KUKA KRL program: G1_Prog.src, G1_Prog.dat

--- G1_Prog.src ---
&ACCESS RVP
DEF  G1_Prog ( )

   GLOBAL INTERRUPT DECL 3 WHEN $STOPMESS==TRUE DO IR_STOPM ( )
   INTERRUPT ON 3
   BAS (#INITMOV,0 )
   BAS (#TOOL, XTOOL)
   BAS (#BASE, XTOOLBASE)

 ;Mover PARA HOME
   SPTP XHOME
   LOOP
      PLC_GET_Pos()
      Gridplace()
      SPTP XHOME
   ENDLOOP

END

DEF PLC_GET_Pos()
   WAIT FOR $IN[19]
   WAIT FOR NOT $IN[19]
   NextPos = 0

   IF $IN[19]THEN
      NextPos=NextPos+1
   ENDIF
   IF $IN[20]THEN
      NextPos=NextPos+2
   ENDIF
   IF $IN[21]THEN
      NextPos=NextPos+4
   ENDIF
   IF $IN[22]THEN
      NextPos=NextPos+8
   ENDIF
END

DEF Gridplace()
   SWITCH NextPos
      CASE 0
         ;insert your code here
         MoveTo(Matrix_Pos1)
      CASE 1
         ;insert your code here
         MoveTo(Matrix_Pos2)
      CASE 2
         ;insert your code here
         MoveTo(Matrix_Pos3)
      CASE 3
         ;insert your code here
         MoveTo(Matrix_Pos4)
      CASE 4
         ;insert your code here
         MoveTo(Matrix_Pos5)
      CASE 5
         ;insert your code here
         MoveTo(Matrix_Pos6)
      CASE 6
         ;insert your code here
         MoveTo(Matrix_Pos7)
      CASE 7
         ;insert your code here
         MoveTo(Matrix_Pos8)
      CASE 8
         ;insert your code here
         MoveTo(Matrix_Pos9)
      DEFAULT
         ;insert your code here
   ENDSWITCH
END

DEF MoveTo(Position:IN)
 POS Position
 RECOLHA.C = 0
 Position.C = 0

 ;IR PARA RECOLHA
 SPTP RECOLHA WITH $VEL_AXIS[1] = SVEL_JOINT(100.0), $TOOL = STOOL2(FBase), $BASE = SBASE(FBase.BASE_NO), $IPO_MODE = SIPO_MODE(FBase.IPO_FRAME), $LOAD = SLOAD(FBase.TOOL_NO), $ACC_AXIS[1] = SACC_JOINT(PPDAT), $APO = SAPO_PTP(PPDAT), $GEAR_JERK[1] = SGEAR_JERK(PPDAT), $COLLMON_TOL_PRO[1] = USE_CM_PRO_VALUES(0) C_Spl
 RECOLHA.Z = RECOLHA.Z - Z_Offset
 LIN RECOLHA
 RECOLHA.C = RECOLHA.C - Angle_Offset
 LIN RECOLHA
 RECOLHA.Z = RECOLHA.Z + Z_Offset
 LIN RECOLHA
 ;RECOLHA.C = RECOLHA.C + Angle_Offset
 ;LIN RECOLHA

 ;IR PARA POSITION
 Position.C = Position.C - Angle_Offset
 SPTP Position WITH $VEL_AXIS[1] = SVEL_JOINT(100.0), $TOOL = STOOL2(FBase), $BASE = SBASE(FBase.BASE_NO), $IPO_MODE = SIPO_MODE(FBase.IPO_FRAME), $LOAD = SLOAD(FBase.TOOL_NO), $ACC_AXIS[1] = SACC_JOINT(PPDAT), $APO = SAPO_PTP(PPDAT), $GEAR_JERK[1] = SGEAR_JERK(PPDAT), $COLLMON_TOL_PRO[1] = USE_CM_PRO_VALUES(0) C_Spl
 Position.Z = Position.Z - Z_Offset
 LIN Position
 Position.C = Position.C + Angle_Offset
 LIN Position
 Position.Z = Position.Z + Z_Offset
 LIN Position
 ;Position.C = Position.C + Angle_Offset
 ;LIN Position

 ;
 RECOLHA.C = RECOLHA.C - Angle_Offset
END

--- G1_Prog.dat ---
&ACCESS RVP
&REL 1
&PARAM DISKPATH = KRC:\R1\Program\Teste G1
DEFDAT  G1_PROG
;FOLD EXTERNAL DECLARATIONS;%{PE}%MKUKATPBASIS,%CEXT,%VCOMMON,%P
;FOLD BASISTECH EXT;%{PE}%MKUKATPBASIS,%CEXT,%VEXT,%P
EXT  BAS (BAS_COMMAND  :IN,REAL  :IN )

DECL INT XTOOLBASE=3 ; ou o n?mero real da sua base
DECL INT XTOOL=3
DECL INT NextPos

DECL INT Z_Offset=50
DECL INT Angle_Offset=45

DECL POS RECOLHA={X -53.7200,Y -200.000,Z 133.000,C -90.0000}
DECL POS Matrix_Pos1={X 100.000,Y 200.000,Z 133.000,C 0.0}
DECL POS Matrix_Pos2={X 20.0000,Y 200.000,Z 133.000,C 0.0}
DECL POS Matrix_Pos3={X -60.0000,Y 200.000,Z 133.000,C 0.0}
DECL POS Matrix_Pos4={X 100.000,Y 120.000,Z 133.000,C 0.0}
DECL POS Matrix_Pos5={X 20.0000,Y 120.000,Z 133.000,C 0.0}
DECL POS Matrix_Pos6={X -60.0000,Y 120.000,Z 133.000,C 0.0}
DECL POS Matrix_Pos7={X 100.000,Y 40.0000,Z 133.000,C 0.0}
DECL POS Matrix_Pos8={X 20.0000,Y 40.0000,Z 133.000,C 0.0}
DECL POS Matrix_Pos9={X -60.0000,Y 40.0000,Z 133.000,C 0.0}


;ENDFOLD (BASISTECH EXT)
;FOLD USER EXT;%{E}%MKUKATPUSER,%CEXT,%VEXT,%P
;Make your modifications here

;ENDFOLD (USER EXT)
;ENDFOLD (EXTERNAL DECLARATIONS)
DECL MODULEPARAM_T LAST_TP_PARAMS={PARAMS[] "Kuka.PointName=Matrix_Pos1; Kuka.FrameData.base_no=2; Kuka.FrameData.tool_no=1; Kuka.FrameData.ipo_frame=#BASE; Kuka.isglobalpoint=False; Kuka.MoveDataName=CPDAT1; Kuka.MovementData.cb={AUX_PT {ORI #CONSIDER,E1 #CONSIDER,E2 #CONSIDER,E3 #CONSIDER,E4 #CONSIDER,E5 #CONSIDER,E6 #CONSIDER},TARGET_PT {ORI #INTERPOLATE,E1 #INTERPOLATE,E2 #INTERPOLATE,E3 #INTERPOLATE,E4 #INTERPOLATE,E5 #INTERPOLATE,E6 #INTERPOLATE}}; Kuka.MovementData.apo_fac=50; Kuka.MovementData.apo_dist=500; Kuka.MovementData.axis_acc=100; Kuka.MovementData.axis_vel=100; Kuka.MovementData.circ_typ=#BASE; Kuka.MovementData.jerk_fac=50; Kuka.MovementData.ori_typ=#VAR; Kuka.MovementData.vel=2; Kuka.MovementData.acc=100; Kuka.MovementData.exax_ign=0; Kuka.VelocityPath=2; Kuka.BlendingEnabled=True; Kuka.APXEnabled=False; Kuka.CurrentCDSetIndex=0; Kuka.VelocityFieldEnabled=False; Kuka.ColDetectFieldEnabled=False; Kuka.MovementParameterFieldEnabled=False; Kuka.IsAngleEnabled=False; Kuka.MoveDataPtpName=PDAT4; Kuka.MovementDataPdat.apo_mode=#CDIS; Kuka.MovementDataPdat.apo_dist=500; Kuka.VelocityPtp=100  "}
DECL PDAT PPDAT={VEL 100.000,ACC 100.000,APO_DIST 500.000,APO_MODE #CDIS,GEAR_JERK 100.000,EXAX_IGN 0}
DECL FDAT FBase={TOOL_NO 3,BASE_NO 3,IPO_FRAME #BASE,POINT2[] " "}

ENDDAT
